// TIA Portal V20 export
// export: Created 2025-12-01T14:56:12.1549484Z, ExportSetting None, DisplayName Totally Integrated Automation Portal, DisplayVersion V20 Update 3, DisplayName TIA Portal Openness, DisplayVersion V20 Update 3, DisplayName TIA Portal Version Control Interface, DisplayVersion V20 Update 3, DisplayName STEP 7 Professional, DisplayVersion V20 Update 3, DisplayName STEP 7 Safety, DisplayVersion V20 Update 2, DisplayName WinCC Basic/Comfort/Advanced, DisplayVersion V20 Update 3, DisplayName WinCC Professional, DisplayVersion V20 Update 3, DisplayName WinCC Unified, DisplayVersion V20 Update 3
TYPE "PulsadorZona"
   STRUCT
      Bit_00 : Bool;
      P_Marcha : Bool;
      P_Rearme : Bool;
      P_TestLuces : Bool;
      P_Auto : Bool := true;
      P_Paro : Bool;
      Bit_06 : Bool;
      Bit_07 : Bool;
      EmergenciaLeve : Bool;
      EmergenciaGrave : Bool;
      ErrorLeve : Bool;
      ErrorGrave : Bool;
      AvisoError : Bool;
      FinReset : Bool;
      MemoriaPulsadorMarcha : Bool;
      MemoriaPulsadorParo : Bool;
   END_STRUCT;
END_TYPE
